INTERFACE ITF_BaseLogger_HMI

END_INTERFACE

(* stored: Version 1.1.0.1
   Itf ITF_BaseLogger_HMI: Id {6de4e498-9c45-0079-3b66-6af767d453b2} *)
